FUNCTION_BLOCK LogSource IMPLEMENTS I_LogSource
VAR
	{attribute 'hide'}
	_SourceName : T_MaxString;
	{attribute 'hide'}
	_Timestamp : T_FILETIME64;
END_VAR

{attribute 'monitoring':='call'}
PROPERTY SourceName : T_MaxString
GET
Sourcename := _Sourcename;
END_GET
SET
_SourceName := SourceName;
END_SET
END_PROPERTY

{attribute 'monitoring':='call'}
PROPERTY Timestamp : T_FILETIME64
GET
Timestamp := _Timestamp;
END_GET
SET
_Timestamp := Timestamp;
END_SET
END_PROPERTY

END_FUNCTION_BLOCK

(* stored: Version 1.1.0.1, ProductVersion 3.1.4026.18
   POU LogSource: Id {832b5691-5c25-458b-b866-144b03f43432}, SpecialFunc None
   Property SourceName: Id {ded94e60-d8cb-4544-89bc-e7b8b1dbd5d8}
   Get Get: Id {0ea29563-228a-4533-971b-c24ed6b53c52}
   Set Set: Id {e5baa9fe-167c-4915-bde8-98944cb4cabf}
   Property Timestamp: Id {592bb9ac-ad7e-482e-8a7e-b468705ce672}
   Get Get: Id {10dd0d44-3088-4d92-990e-2f1c8113c1c1}
   Set Set: Id {e5bdbf5e-1d3b-4d67-97b7-bc3d87863e45} *)
